(* PLC project Unnamed, Unknown Unnamed 1 *)
(* stored: creationDateTime 2020-09-15T10:36:20, modificationDateTime 2021-08-28T20:33:24 *)

PROGRAM part1b
  VAR
    Input0 AT %IX1.0 : BOOL;
    Output0 AT %QX1.0 : BOOL;
  END_VAR
  VAR
    Oscillator : BOOL;
    TON0 : TON;
    TOF0 : TOF;
  END_VAR

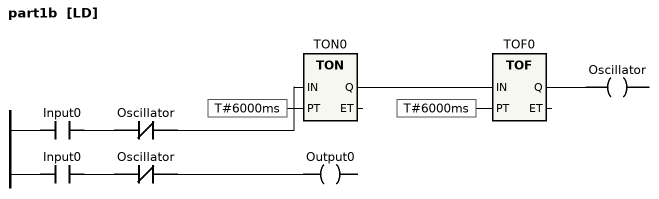
(* LD diagram, written out as Structured Text *)
TON0(IN := Input0 AND NOT Oscillator, PT := T#6000ms);
TOF0(IN := TON0.Q, PT := T#6000ms);
Oscillator := TOF0.Q;
Output0 := Input0 AND NOT Oscillator;
END_PROGRAM

CONFIGURATION Config0
  RESOURCE Res0 ON PLC
    TASK task0(INTERVAL := T#20ms, PRIORITY := 0);
    PROGRAM instance0 WITH task0 : part1b;
  END_RESOURCE
END_CONFIGURATION
